FUNCTION_BLOCK KukaRobot
VAR_OUTPUT
	forceStop AT %Q* : BOOL;
	resetSignal AT %Q* : BOOL;
	
	outputs AT %Q* : ARRAY[1..50] OF INT;
	inputs AT %I* : ARRAY[1..20] OF INT;
	
	taskID : INT;
	completedTask : INT;
	
	operational : BOOL;
	reserved : BOOL;
	reservation : SectionEnum := SectionEnum.NULL_SECTION;
	tool : SectionEnum := SectionEnum.WOOD_BUNK;
	
	error : BOOL;
	errId : DINT;
END_VAR
VAR
	step : (SEND_COMMAND, WAIT);
END_VAR

taskID := outputs[1];
completedTask := inputs[1];

{attribute 'monitoring' := 'variable'}
{attribute 'monitoring' := 'call'}
PROPERTY Busy : BOOL
GET
VAR
	emptyOutput : ARRAY[1..50] OF INT;
END_VAR

//Busy stays TRUE until outputs are cleared AND completed task has elapsed
//Ready is always inverse of Busy
updateStatus();

Busy :=
	MEMCMP(ADR(outputs), ADR(emptyOutput), SIZEOF(outputs)) <> 0 OR
	completedTask <> 0;
END_GET
END_PROPERTY

METHOD commandEx : BOOL
VAR_INPUT
	newOutputs : REFERENCE TO ARRAY[1..50] OF INT;
END_VAR
outputs := newOutputs;
END_METHOD

//{attribute 'monitoring' := 'variable'}
{attribute 'monitoring' := 'call'}
PROPERTY Done : BOOL
GET
updateStatus();

Done := completedTask = taskID;
END_GET
END_PROPERTY

METHOD eStop : BOOL
VAR_INPUT
END_VAR
forceStop := TRUE;
eStop := TRUE;
END_METHOD

METHOD idleCommand : BOOL
VAR_INPUT
END_VAR
MEMSET(ADR(outputs), 0, SIZEOF(outputs));
END_METHOD

PROPERTY Ready : BOOL
GET
updateStatus();

Ready := NOT Busy;
END_GET
END_PROPERTY

METHOD release : BOOL
VAR_INPUT
	sectionReservation : SectionEnum;
END_VAR
IF reservation = sectionReservation AND reserved THEN
	reservation := SectionEnum.NULL_SECTION;
	reserved := FALSE;
	release := TRUE;
END_IF
END_METHOD

METHOD reserve : BOOL
VAR_INPUT
	reserveRequest : SectionEnum;
END_VAR
(*
this method exists because chipboard and wood bunk operations use the same robot
both sections need to check if the robot is open to commands before use
*)
IF reserved AND reservation = reserveRequest THEN
	reserve := TRUE;

ELSIF (NOT reserved) AND reservation = SectionEnum.NULL_SECTION THEN
	reservation := reserveRequest;
	reserved := TRUE;
	reserve := TRUE;

END_IF
END_METHOD

METHOD reset : BOOL
//resetSignal := TRUE;
//done := FALSE;

MEMSET(ADR(outputs), 0, SIZEOF(outputs));
(*
IF ready AND completedTask = 0 THEN
	resetSignal := FALSE;
	reset := TRUE;
END_IF
*)
END_METHOD

METHOD resume : BOOL
VAR_INPUT
END_VAR
forceStop := FALSE;

resume := NOT error AND errId = 0;
END_METHOD

METHOD setCommandAndWait : BOOL
VAR_INPUT
	newOutputs : REFERENCE TO ARRAY[1..50] OF INT;
END_VAR
//IF NOT Busy THEN
	//RETURN;
//END_IF

outputs := newOutputs;
setCommandAndWait := Done;

(*
CASE step OF
	SEND_COMMAND: //wait 1 cycle
		outputs := newOutputs;
		step := WAIT;
		
	WAIT:
		IF done THEN
			(*	
			IF NOT reset() THEN
				RETURN;
			END_IF
			
			step := 0;
			*)
			setCommandAndWait := TRUE;
		END_IF
		
END_CASE
*)
END_METHOD

METHOD updateStatus : BOOL
VAR_INPUT
END_VAR
taskID := outputs[1];
completedTask := inputs[1];
END_METHOD

END_FUNCTION_BLOCK

(* stored: Version 1.1.0.1, ProductVersion 3.1.4024.11
   POU KukaRobot: Id {870b17d8-8fed-45ea-b532-f3f727b3e8ec}, SpecialFunc None
   Folder Properties: Id {866be447-1963-4a08-8cb7-28bb42cb4605}
   Property Busy: Id {b3d2dd20-1b64-42bd-b7b9-cc40de53165e}
   Get Get: Id {3bf870ef-0c1b-46d6-841d-b325e44d6211}
   Method commandEx: Id {55c20752-492d-4e9a-a647-f2d920916f43}
   Property Done: Id {aab115a2-23cb-4864-ae41-4499fdda0c27}
   Get Get: Id {f35a7b96-3469-4c48-a415-04be19290868}
   Method eStop: Id {974b2363-087f-4f71-a37b-fdee6dacfa65}
   Method idleCommand: Id {4f96fde8-b481-408a-8e4e-1ca7d5a2c9bb}
   Property Ready: Id {b09b77a8-11f4-47fb-9077-e4f375d271da}
   Get Get: Id {86e66399-49b2-4e73-8b04-ebe19b5e9e41}
   Method release: Id {7fed4361-8a94-445d-8040-f071f846d639}
   Method reserve: Id {1e01deef-588d-4739-a104-23ce337539cb}
   Method reset: Id {89eb6678-027f-45a1-a94f-ae23b58ecc5c}
   Method resume: Id {1d12dfe1-c8ff-4b57-9b31-0d4b08a72b4a}
   Method setCommandAndWait: Id {861e79f4-9d73-4326-81bf-3ad217fcca64}
   Method updateStatus: Id {fb027fa2-67ff-4c87-b192-f170e88fa5be} *)
